// TIA Portal V17 export
// export: Created 2025-06-25T13:13:12.1863745Z, ExportSetting WithDefaults, DisplayName Totally Integrated Automation Portal, DisplayVersion V17 Update 8, DisplayName TIA Portal Openness, DisplayVersion V17 Update 8, DisplayName TIA Portal Version Control Interface, DisplayVersion V17, DisplayName STEP 7 Professional, DisplayVersion V17 Update 8, DisplayName STEP 7 Safety, DisplayVersion V17 Update 6, DisplayName WinCC Advanced, DisplayVersion V17 Update 8
DATA_BLOCK "StateMachine_DB"   // DB31
VERSION : 0.1
// stored: AutoNumber true, DBAccessibleFromOPCUA true, DBAccessibleFromWebserver true, InstanceOfName StateMachine, InstanceOfType FB
"StateMachine"
   // VAR
   //    StateChanges : Struct
   //       "0-zu-1_StateChange" : Bool;
   //       "1-zu-2_StateChange" : Bool;
   //       "2-zu-3_StateChange" : Bool;
   //       "2-zu-7_StateChange" : Bool;
   //       "3-zu-2_StateChange" : Bool;
   //       "3-zu-4_StateChange" : Bool;
   //       "3-zu-7_StateChange" : Bool;
   //       "4-zu-2_StateChange" : Bool;
   //       "4-zu-5_StateChange" : Bool;
   //       "4-zu-7_StateChange" : Bool;
   //       "5-zu-2_StateChange" : Bool;
   //       "5-zu-6_StateChange" : Bool;
   //       "5-zu-7_StateChange" : Bool;
   //       "6-zu-2_StateChange" : Bool;
   //       "6-zu-7_StateChange" : Bool;
   //       "7-zu-1_StateChange" : Bool;
   //    END_STRUCT;
   //    Evaluate_DB : "Evaluate";
   // END_VAR
BEGIN
END_DATA_BLOCK
